{attribute 'GeneratedUsingTerminal: IODEVICETYPE_ETHERCATPROT'}
{attribute addProperty BoxType "IODEVICETYPE_ETHERCATPROT"}
{attribute addProperty Id "Term_1_EK1100Term_1_EK1100_C62D072D20SyncUnitsSyncUnits_99E584AF18InputsInputs_A65FACA410OutputsOutputs_23C0ED1D6InfoDataInfoData_C76BEFB322"}
{attribute addProperty CRC "3693654007"}
{attribute addProperty Size "76"}
TYPE Device_1_EtherCAT_DC28AFF7 :
STRUCT
	{attribute addProperty Name "Term_1_EK1100"}
	{attribute addProperty PreviousPort "Device 1 (EtherCAT) : Master"}
	Term_1_EK1100 : Term_1_EK1100_C62D072D;
	{attribute addProperty Name "SyncUnits"}
	SyncUnits : SyncUnits_99E584AF;
	{attribute addProperty Name "Inputs"}
	Inputs : Inputs_A65FACA4;
	{attribute addProperty Name "Outputs"}
	Outputs : Outputs_23C0ED1D;
	{attribute addProperty Name "InfoData"}
	InfoData : InfoData_C76BEFB3;
END_STRUCT
END_TYPE

(* stored: Version 1.2.0.0, ProductVersion 3.1.4024.9
   DUT Device_1_EtherCAT_DC28AFF7: Id {d9cdc395-bd30-468d-b11e-92e721dab65a} *)
